FUNCTION_BLOCK F_DELETE (* delete L characters of IN beginning at the P-th character position *)
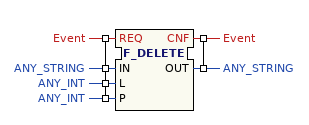
  EVENT_INPUT
    REQ WITH IN, L, P; (* Service Request *)
  END_EVENT
  EVENT_OUTPUT
    CNF WITH OUT; (* Confirmation of Requested Service *)
  END_EVENT
  VAR_INPUT
    IN : ANY_STRING; (* input string *)
    L : ANY_INT; (* length to delete *)
    P : ANY_INT; (* delete start position *)
  END_VAR
  VAR_OUTPUT
    OUT : ANY_STRING; (* substring *)
  END_VAR
END_FUNCTION_BLOCK
